// TIA Portal V20 export
VAR_GLOBAL   // PLC tag table "Unit1"
   "BA040AZSSP201.00" AT %I700.0 : Bool;   // AUTO INITIATE PBL (GREEN)
   "BA040AZSSP201.01" AT %I700.1 : Bool;   // STOP PBL (RED)
   "BA040AZSSP201.10" AT %I701.0 : Bool;   // MAIN HMI POWER TRIPPED E110CB
   "BA040AZSSP501.00" AT %I3000.0 : Bool;   // CONTROL DC POWER TRIPPED E156CB
   "BA040AZSSP501.01" AT %I3000.1 : Bool;   // SAFETY DC POWER TRIPPED E218CB
   "BA040AZSSP501.02" AT %I3000.2 : Bool;   // CLASS 2 SMPS POWER TRIPPED E308CB
   "BA040AZSSP501.03" AT %I3000.3 : Bool;   // CLASS 2 SMPS MONITORING E310PWS
   "BA040AZSSP501.04" AT %I3000.4 : Bool;   // ET200ECO PN-1 POWER TRIPPED E324CB
   "BA040AZSSP501.05" AT %I3000.5 : Bool;   // ET200ECO PN-2 POWER TRIPPED E328CB
   "BA040AZSSP501.06" AT %I3000.6 : Bool;   // ET200ECO PN-3 POWER TRIPPED E332CB
   "BA040AZSSP501.07" AT %I3000.7 : Bool;   // ET200ECO PN-4 POWER TRIPPED E336CB
   "BA040AZSSP202.00" AT %Q700.0 : Bool;   // MAIN OP AUTO INITIATE PBL LAMP ON (GREEN)
   "BA040AZSSP202.01" AT %Q700.1 : Bool;   // MAIN OP STOP PBL LAMP ON (RED)
   "BA040AZSSP202.03" AT %Q700.3 : Bool;   // MAIN OP ENABLE PBL LAMP ON (WHITE)
   "BA040AZSSP202.04" AT %Q700.4 : Bool;   // MAIN OP SAFETY RESET PBL LAMP ON (BLUE)
   "BA040AZSSP202.12" AT %Q701.2 : Bool;   // TOWER LAMP 3 ON (GREEN)
   "BA040AZSSP202.13" AT %Q701.3 : Bool;   // TOWER LAMP 4 ON (WHITE)
   "BA040AZSSP202.14" AT %Q701.4 : Bool;   // TOWER LAMP 5 ON (BLUE)
   "BA040AZSSP502.00" AT %Q3000.0 : Bool;   // CLASS2 SMPS ALARM RESET
   BA040AZSCU1_Actor_Interface_AddressIn AT %I5000.0 : "LPD_typePDTel390In";
   BA040AZSCU1_Actor_Interface_AddressOut AT %Q5000.0 : "LPD_typePDTel390Out";
   BA040AZSCU2_Actor_Interface_AddressIn AT %I5004.0 : "LPD_typePDTel390In";
   BA040AZSCU2_Actor_Interface_AddressOut AT %Q5004.0 : "LPD_typePDTel390Out";
   BA040AZSCU3_Actor_Interface_AddressIn AT %I5008.0 : "LPD_typePDTel390In";
   BA040AZSCU3_Actor_Interface_AddressOut AT %Q5008.0 : "LPD_typePDTel390Out";
   BA040AZSCU4_Actor_Interface_AddressIn AT %I5012.0 : "LPD_typePDTel390In";
   BA040AZSCU4_Actor_Interface_AddressOut AT %Q5012.0 : "LPD_typePDTel390Out";
   BA040AZSCU5_Actor_Interface_AddressIn AT %I5016.0 : "LPD_typePDTel390In";
   BA040AZSCU5_Actor_Interface_AddressOut AT %Q5016.0 : "LPD_typePDTel390Out";
   BA040AZSCU6_Actor_Interface_AddressIn AT %I5020.0 : "LPD_typePDTel390In";
   BA040AZSCU6_Actor_Interface_AddressOut AT %Q5020.0 : "LPD_typePDTel390Out";
   BA040AZSCU7_Actor_Interface_AddressIn AT %I5024.0 : "LPD_typePDTel390In";
   BA040AZSCU7_Actor_Interface_AddressOut AT %Q5024.0 : "LPD_typePDTel390Out";
   BA040AZSCU8_Actor_Interface_AddressIn AT %I5028.0 : "LPD_typePDTel390In";
   BA040AZSCU8_Actor_Interface_AddressOut AT %Q5028.0 : "LPD_typePDTel390Out";
   BA040AZSCU9_Actor_Interface_AddressIn AT %I5032.0 : "LPD_typePDTel390In";
   BA040AZSCU9_Actor_Interface_AddressOut AT %Q5032.0 : "LPD_typePDTel390Out";
   BA040AZSSLM1_Actor_Interface_AddressIn AT %I5050.0 : "LPD_typePDTel370In";
   BA040AZSSLM1_Actor_Interface_AddressOut AT %Q5050.0 : "LPD_typePDTel370Out";
   "BA040AZSMP101.02" AT %I100.2 : Bool;   // E6404PWS CONTROLLER POWER SMPS AC POWER TRIPPED E214CB
   "BA040AZSMP101.03" AT %I100.3 : Bool;   // E6704PWS CONTROLLER POWER SMPS AC POWER TRIPPED E222CB
   "BA040AZSMP101.04" AT %I100.4 : Bool;   // E6804PWS SAFETY POWER SMPS AC POWER TRIPPED E226CB
   "BA040AZSMP101.06" AT %I100.6 : Bool;   // PROCESSOR POWER ON TIPPRED E4120CB
   "BA040AZSMP101.07" AT %I100.7 : Bool;   // PROGRAMING POWER OUTLET TRPPED E4126CB
   "BA040AZSMP101.11" AT %I101.1 : Bool;   // PANEL LED POWER TRIPPED E4304CB
   "BA040AZSMP101.13" AT %I101.3 : Bool;   // PLC POWER SMPS DC OK E4404PWS
   "BA040AZSMP101.14" AT %I101.4 : Bool;   // CONTROL LEVEL HUB POWER TRIPPED E4420CB
   "BA040AZSMP101.15" AT %I101.5 : Bool;   // MAIN HMI POWER TRIPPED E4426CB
   "BA040AZSMP101.16" AT %I101.6 : Bool;   // PORTABLE HMI POWER TIPPED E4432CB
   "BA040AZSMP101.17" AT %I101.7 : Bool;   // PANEL IRT HUB POWER TIPPED E4604CB
   "BA040AZSMP101.20" AT %I102.0 : Bool;   // IRT HUB FAULT E4608ES
   "BA040AZSMP101.23" AT %I102.3 : Bool;   // 120VAC CONTROL POWER TR SECONDARY TRIPPED E5110CB
   "BA040AZSMP101.24" AT %I102.4 : Bool;   // CONTROL POWER ON TRIPPED E5120CB
   "BA040AZSMP101.25" AT %I102.5 : Bool;   // VISION MONITOR-1&MCU POWER STRIP OUTLET POWER TRIPPED E5126CB
   "BA040AZSMP101.26" AT %I102.6 : Bool;   // VISION MONITOR-2&VISION MONITOR-3 POWER STRIP OUTLET POWER TRIPPED E5132CB
   "BA040AZSMP101.27" AT %I102.7 : Bool;
   "BA040AZSMP101.31" AT %I103.1 : Bool;   // FFU POWER-1 POWER TRIPPED E5222CB
   "BA040AZSMP101.33" AT %I103.3 : Bool;   // CONTROL POWER SMPS DC OK E6104PWS
   "BA040AZSMP101.34" AT %I103.4 : Bool;   // ET200MP I/O OUTPUT POWER TRIPPED E6154CB
   "BA040AZSMP101.35" AT %I103.5 : Bool;   // JUNCTION BOX CONTROL POWER TRIPPED E6180CB
   "BA040AZSMP101.36" AT %I103.6 : Bool;   // CLASS 2 SMPS POWER TRIPPED E6204CB
   "BA040AZSMP101.37" AT %I103.7 : Bool;   // CLASS 2 SMPS MONITORING E6206PWS
   "BA040AZSMP102.00" AT %I104.0 : Bool;   // ET200ECO PN-1 POWER TRIPPED E6220CB
   "BA040AZSMP102.01" AT %I104.1 : Bool;   // ET200ECO PN-2 POWER TRIPPED E6224CB
   "BA040AZSMP102.02" AT %I104.2 : Bool;   // ET200ECO PN-3 POWER TRIPPED E6228CB
   "BA040AZSMP102.03" AT %I104.3 : Bool;   // ET200ECO PN-4 POWER TRIPPED E6232CB
   "BA040AZSMP102.04" AT %I104.4 : Bool;   // PANEL FAN POWER TRIPPED E6304CB
   "BA040AZSMP102.06" AT %I104.6 : Bool;   // CONTROLLER POWER SMPS DC OK E6404PWS
   "BA040AZSMP102.07" AT %I104.7 : Bool;   // CONTROLLER DC POWER TRIPPED E6406CB
   "BA040AZSMP102.11" AT %I105.1 : Bool;   // MANIFOLD-1 CONTROL POWER TRIPPED E6422CB
   "BA040AZSMP102.12" AT %I105.2 : Bool;   // MANIFOLD-2 CONTROL POWER TRIPPED E6430CB
   "BA040AZSMP102.13" AT %I105.3 : Bool;   // DRIVE-CLIQ HUB POWER TRIPPED E6456CB
   "BA040AZSMP102.14" AT %I105.4 : Bool;   // DRIVE-CLIQ HUB POWER TRIPPED E6462CB
   "BA040AZSMP102.15" AT %I105.5 : Bool;   // HANDY QR READER POWER TRIPPED E6468CB
   "BA040AZSMP102.16" AT %I105.6 : Bool;   // VISION CONTROLLER-1 POWER TRIPPED E6474CB
   "BA040AZSMP102.17" AT %I105.7 : Bool;   // VISION CONTROLLER-2 POWER TRIPPED E6480CB
   "BA040AZSMP102.20" AT %I106.0 : Bool;   // VISION CONTROLLER-3 POWER TRIPPED E6486CB
   "BA040AZSMP102.21" AT %I106.1 : Bool;   // LINE LASER MODULE-1 POWER TRIPPED E6506CB
   "BA040AZSMP102.22" AT %I106.2 : Bool;   // LINE LASER MODULE-2 POWER TRIPPED E6512CB
   "BA040AZSMP102.24" AT %I106.4 : Bool;   // CONTROLLER POWER SMPS DC OK E6704PWS
   "BA040AZSMP102.25" AT %I106.5 : Bool;   // CONTROLLER DC POWER TRIPPED E6706CB
   "BA040AZSMP102.26" AT %I106.6 : Bool;   // EPC CONTROLLER-1 POWER TRIPPED E6716CB
   "BA040AZSMP102.27" AT %I106.7 : Bool;   // EPC CONTROLLER-2 POWER TRIPPED E6722CB
   "BA040AZSMP102.30" AT %I107.0 : Bool;   // EPC CONTROLLER-3 POWER TRIPPED E6728CB
   "BA040AZSMP102.31" AT %I107.1 : Bool;   // EPC CONTROLLER-4 POWER TRIPPED E6734CB
   "BA040AZSMP102.32" AT %I107.2 : Bool;   // SAFETY POWER SMPS DC OK E6804PWS
   "BA040AZSMP102.33" AT %I107.3 : Bool;   // SAFETY DC POWER TRIPPED E6806CB
   "BA040AZSMP102.34" AT %I107.4 : Bool;   // ET200SP I/O SAFETY POWER TRIPPED E6816CB
   "BA040AZSMP102.35" AT %I107.5 : Bool;   // JUNCTION BOX CONTROL POWER TRIPPED E6836CB
   "BA040AZSMP102.36" AT %I107.6 : Bool;   // ET200ECO PN SAFETYT-1 POWER TRIPPED E6856CB
   "BA040AZSMP102.37" AT %I107.7 : Bool;   // ET200ECO PN SAFETYT-2 POWER TRIPPED E6862CB
   "BA040AZSMP104.03" AT %Q100.3 : Bool;   // CLASS2 SMPS ALARM RESET
   "BA040AZSSP202.10" AT %Q701.0 : Bool;   // TOWER LAMP 1 ON (RED)
   "BA040AZSSP202.11" AT %Q701.1 : Bool;   // TOWER LAMP 2 ON (AMBER)
   "BA040AZSSP202.15" AT %Q701.5 : Bool;   // TOWER LAMP BUZZER ON
   "BA040AZSMP104.11" AT %Q101.1 : Bool;   // SPARE
   "BA040AZSMP104.12" AT %Q101.2 : Bool;   // SPARE
   "BA040AZSMP104.13" AT %Q101.3 : Bool;   // SPARE
   "BA040AZSMP104.14" AT %Q101.4 : Bool;   // SPARE
   "BA040AZSMP103.00" AT %I108.0 : Bool;   // DC-DC CONVERTER IN POWER TRIPPED E6756CB
   "BA040AZSMP103.01" AT %I108.1 : Bool;   // HOT WIRE CUTTER POWER TRIPPED E6762CB
   "BA040AZSMP103.04" AT %I108.4 : Bool;   // SPARE
   "BA040AZSMP103.06" AT %I108.6 : Bool;   // SPARE
   "BA040AZSBK26.02" AT %I1100.2 : Bool;   // MAIN VALVE DIGITAL PRESSURE SWITCH OUT1
   "BA040AZSBK26.12" AT %I1101.2 : Bool;   // MAIN VALVE DIGITAL PRESSURE SWITCH OUT2
END_VAR
VAR_GLOBAL CONSTANT   // user constants
   U1_NO_OF_EMs : Int := 7;   // Highest Value of equipment modules in the unit (Counting starts from 0)
   U1_EM0 : Int := 0;
   U1_EM1 : Int := 1;
   U1_EM2 : Int := 2;
   U1_EM3 : Int := 3;
   U1_EM4 : Int := 4;
   U1_EM5 : Int := 5;
   U1_EM6 : Int := 6;
   U1_EM7 : Int := 7;
   U1_NO_OF_PARTPLACE : Int := 9;
   U1_EM6_TRACKING_Count : UInt := 60;
   U1_EM4_GageRR_Count : UInt := 60;
   U1_EM5_GageRR_Count : UInt := 60;
END_VAR
